GLOBALCONSTANTS START (* Global constants *)
  (* Standard: 61499-1 *)
  (* Version 1.0, 2025-05-23, franz *)
  PACKAGE Schieber::AufZu;
  VAR_GLOBAL CONSTANT
    Closed : UINT := UINT#5;
    Opened : UINT := UINT#6;
    Unknown : UINT := UINT#7;
  END_VAR
END_GLOBALCONSTANTS
